// Mitsubishi GX Works2 project: finalfinal   PLC: FX3G

// global labels: Global1
VAR_GLOBAL
  workDayLight AT Y010 : BOOL;  (* Y010 is the work day light- lighting while the day running *)
  emergencyButton AT X007 : BOOL;  (* emergency button when click on the day stop *)
  startBlink AT M0 : BOOL;  (* when click on X007 -emergency button- the blinking function starts *)
  monitoringLighter AT M1 : BOOL;  (* monitoring light of the blinking *)
  timerBlink1 AT TC1 : BOOL;  (* timer for blink every 1 sec *)
  endTimerBlink1 AT TS1 : BOOL;  (* get value of 1 when TC1 is ending *)
END_VAR
VAR_GLOBAL CONSTANT
  timeBlink1 : INT := 10;
END_VAR
VAR_GLOBAL
  blinkLight1 AT M2 : BOOL;  (* one of the two lights that blinking in the blinking function that light Y010 blinking *)
  timerBlink2 AT TC2 : BOOL;  (* timer for blink every 1 sec *)
END_VAR
VAR_GLOBAL CONSTANT
  timeBlink2 : INT := 10;
END_VAR
VAR_GLOBAL
  endTimerBlink2 AT TS2 : BOOL;  (* get value of 1 when TC2  is ending *)
  blinkLight2 AT M3 : BOOL;  (* one of the blinking bulbs *)
END_VAR
VAR_GLOBAL CONSTANT
  initializeOrange : REAL := 170;  (* orange input for orit *)
END_VAR
VAR_GLOBAL
  startDayFictiveLight AT M4 : BOOL;  (* one condition of start the day- click on X010 start it *)
  stopAfter3Sec AT M5 : BOOL;  (* the light represent the end of 3 sec counting *)
END_VAR
VAR_GLOBAL CONSTANT
  count3Sec : INT := 600;
END_VAR
VAR_GLOBAL
  count3Sec2 AT TS3 : BOOL;  (* get 1 when TC3 ends after 3 sec *)
END_VAR
VAR_GLOBAL CONSTANT
  timer3Sec : INT := 30;
END_VAR
VAR_GLOBAL
  counter3Sec AT TC3 : BOOL;  (* 3 sec count for 2 bulbs blink 3 sec only and then stop *)
  orangeInput AT D1119 : REAL;  (* the amount of oranges we get for input *)
  OrangeQuantity AT D1121 : REAL;  (* moving orange input to our orange stack *)
  clementineInput AT D1123 : REAL;  (* the amount of clementine we get for input *)
  clementineQuantity AT D1125 : REAL;  (* moving clementine input to our clementine stack *)
  pomeloInput AT D1127 : REAL;  (* the amount of pomelo we get for input *)
  pomeloQuantity AT D1129 : REAL;  (* moving pomelo input to our pomelo stack *)
END_VAR
VAR_GLOBAL CONSTANT
  minOrange : REAL := 2.0;  (* check if we have at least 2 oranges unless the day cannot start *)
  minClementine : REAL := 1.0;  (* check if we have at least 1 clementine unless the day cannot start *)
  minPomelo : REAL := 1.0;  (* check if we have at least 1 pomelo unless the day cannot start *)
END_VAR
VAR_GLOBAL
  componentTesting AT M15 : BOOL;  (* if all the conditions are true the day can start *)
END_VAR
VAR_GLOBAL CONSTANT
  constantRatio : REAL := 2.0;  (* deviding or double orange in 2 *)
END_VAR
VAR_GLOBAL
  change AT D1133 : REAL;  (* the minimum of 0.5*orange, clementine, pomelo to use in the iteration *)
  changeOrange AT D1135 : REAL;  (* the real amount of orange we take to iteration *)
END_VAR
VAR_GLOBAL CONSTANT
  maxOrange : REAL := 50;  (* the max orange in iteration can be 100. so, if 0.5*orange is greater then 50 we take 50 *)
  value_1 : REAL := 1;
END_VAR
VAR_GLOBAL
  clemntineToUse AT D1137 : REAL;  (* move the chosen clementine value to use to the variable to use in the iteration *)
  pomeloToUse AT D1139 : REAL;  (* move the chosen pomelo value to use to the variable to use in the iteration *)
  orangeToUse AT D1141 : REAL;  (* move the chosen orange value to use to the variable to use in the iteration *)
  stratWashing AT X002 : BOOL;  (* start washing operation *)
  counter3secWash AT TC4 : BOOL;  (* count 3 sec of Y005 light in the wash operation *)
  washCounter3 AT TS4 : BOOL;  (* get 1 when TC4 3 sec ends *)
  stopLightWashing AT Y005 : BOOL;  (* washing light- light for 3 sec in the wash operation *)
  startWashing AT X002 : BOOL;  (* when part 1 is starting *)
  washingClemintine AT D1143 : REAL;  (* the clementine in the washing machine *)
  washingPomelo AT D1145 : REAL;  (* the pomelo in the washing machine *)
  washingOrange AT D1147 : REAL;  (* the orange in the washing machine *)
  squizeButton AT X001 : BOOL;  (* starts the squize operation *)
  squzeContainer AT D1149 : REAL;  (* all fruites dedicated to squize in the pre squize container *)
  finishWash AT M16 : BOOL;  (* represent the end of washing operation *)
  squizeLightStore AT Y001 : BOOL;  (* squize operation light- light until operation finish *)
  startSquize AT X011 : BOOL;  (* when push it twice the squize operatin starts *)
END_VAR
VAR_GLOBAL CONSTANT
  pushingCounter : INT := 2;
END_VAR
VAR_GLOBAL
  pushingCounterDevice AT CC0 : BOOL;  (* how much times we need to push to start squize *)
  doneCounter AT CS0 : BOOL;  (* when counter done finish squize *)
  squizeLight1 AT Y002 : BOOL;  (* blinking while squizing *)
  squizeLight2 AT Y003 : BOOL;  (* blinking while squizing *)
  emergencyButtonLight AT M8 : BOOL;  (* fictive light for emergency *)
  juiceContainer AT D1151 : REAL;  (* the juice container *)
  finishColectFruits AT M17 : BOOL;  (* when the colect ftuits is done the fictive lamp will light *)
  donesquizeLight AT M19 : BOOL;  (* squize ended *)
  startqualityCheck AT X003 : BOOL;  (* starts quality check operation *)
  startingQAcheckLight AT M20 : BOOL;  (* starting QA check Light *)
END_VAR
VAR_GLOBAL CONSTANT
  lowerBound : REAL := 1.0;  (* lower Bound *)
  upperBound : REAL := 5.0;  (* upper bound *)
END_VAR
VAR_GLOBAL
  timerOfQA AT TC6 : BOOL;  (* timer 5 sec of QA check *)
END_VAR
VAR_GLOBAL CONSTANT
  valueTimerQA : INT := 50;  (* valueTimerQA 5 SEC *)
END_VAR
VAR_GLOBAL
  doneTimerQA AT TS6 : BOOL;  (* when QA GOOD 5 sec light *)
  QAgoodLight AT Y004 : BOOL;  (* when QA GOOD 5 sec light Y005 *)
  stackcontainer AT D1155 : REAL;  (* stack Container *)
  analog_input_2 AT D8281 : INT;
  qualityChecking AT D1163 : REAL;  (* the quality check *)
  ifQAGood AT M22 : BOOL;  (* if QA good *)
  finishedQACheckLight AT M24 : BOOL;  (* when the good juice moved to stack the lamp will light *)
  juiceIsRotenLight AT M23 : BOOL;  (* when the qa check isnt good in the second time the juise is thrown out *)
  finishThrowJuiceLight AT M25 : BOOL;  (* when the roten juice is thrown out the lamp will light *)
  count2switchs AT CC1 : BOOL;  (* get 1 when X3 is up twice *)
END_VAR
VAR_GLOBAL CONSTANT
  twoSwitches : INT := 2;  (* 1 when there are 2 switch ups *)
END_VAR
VAR_GLOBAL
  counter2switches AT CS1 : BOOL;  (* 1 when 2 swiches happened *)
  startBottlingPart AT X005 : BOOL;  (* starts bottling part *)
  bottlingInProcessLight AT Y011 : BOOL;  (* the lamp will light till the bottling is in process *)
END_VAR
VAR_GLOBAL CONSTANT
  minNumOfLiters : REAL := 2.0;  (* check if we have at least 2 liter *)
  twoLittersInBottle : REAL := 2.0;  (* our buttles contains two litters *)
  maxBottles : REAL := 100.0;  (* the maximu bottles we can transfer *)
END_VAR
VAR_GLOBAL
  analog_output AT D8282 : INT;  (* analog value *)
END_VAR
VAR_GLOBAL CONSTANT
  normalizetion : REAL := 408;  (* analog value normalizetion *)
  normalizetion2 : REAL := 408;  (* analog value normalizetion *)
END_VAR
VAR_GLOBAL
  finishFirstBottling AT M6 : BOOL;  (* when the first bottling is done *)
  finishIteration AT Y006 : BOOL;  (* when the iteration is done *)
  timeBeforeSeceondTrack AT TC8 : BOOL;  (* stand still time before track num.2 *)
END_VAR
VAR_GLOBAL CONSTANT
  timeHold : INT := 20;
END_VAR
VAR_GLOBAL
  waitingSwitch AT TS8 : BOOL;  (* waiting for time to end to out track number 2 *)
  newStackContainer AT D1167 : REAL;
  updateInput AT M7 : BOOL;  (* update the input after every iteration *)
  endDay AT M9 : BOOL;  (* emergency button dtart the end day process *)
END_VAR
VAR_GLOBAL CONSTANT
  fourSecHolding : INT := 60;
END_VAR
VAR_GLOBAL
  trackDrivingFor4Sec2 AT TC10 : BOOL;  (* track light working for 4 sec *)
  trackDrivingTimer AT TS10 : BOOL;  (* track light working for 4 sec *)
  squizeStageLight AT X001 : BOOL;  (* squize operation light *)
  squizeStageLight2 AT M10 : BOOL;  (* squize operation light *)
  end5Stage AT M18 : BOOL;  (* indicte that the bottling process is done *)
  endOfBottlingPro AT M11 : BOOL;  (* indicte that the bottling process is done *)
END_VAR
VAR_GLOBAL CONSTANT
  minBottles : REAL := 1.0;  (* check if we have at least 1 clementine unless the day cannot start *)
  endOfBottle : REAL;  (* indicte that the bottling process is done *)
END_VAR
VAR_GLOBAL
  trackLight AT M12 : BOOL;  (* light of end track stage *)
  end5light AT M26 : BOOL;  (* indicte that the bottling process is done *)
  waitingBeforeExit AT TC9 : BOOL;  (* waiting for time to end to out track number 2 *)
  isWaitingOver AT TS9 : BOOL;  (* waiting for time to end to out track number 2 *)
  startSecondtrack AT X011 : BOOL;  (* when push it twice the squize operatin starts *)
  track2Timer AT TC10 : BOOL;  (* track light working for 4 sec *)
  track2Bool AT TS10 : BOOL;  (* track light working for 4 sec *)
  factiveBottlingLight AT M13 : BOOL;  (* gets 1 when bottling proccess start *)
  factiveQALight AT M21 : BOOL;  (* gets 1 when QA ends *)
END_VAR
VAR_GLOBAL CONSTANT
  zero : REAL;  (* zero value *)
END_VAR
VAR_GLOBAL
  factiveY5 AT M30 : BOOL;  (* when Y5 turn on *)
  factiveY1 AT M31 : BOOL;  (* when Y1 turn on *)
  tracl2bool AT TS10 : BOOL;  (* track light working for 4 sec *)
  stackcontainer2 AT D1165 : REAL;  (* stack Container *)
  moveToStackCon AT M27 : BOOL;  (* move stock to new container *)
  endDayZero AT M28 : BOOL;  (* if one of quantities is 0 the day over *)
  endDayZeroHold AT M29 : BOOL;  (* end Day Zero Hold STAY *)
  startDay AT X010 : BOOL;  (* the button for starting a work day *)
  numofBottles AT D1180 : REAL;  (* the new num of the bottles *)
  numofBottlesNew AT D1182 : REAL;  (* the new num of the bottles *)
  enoughFruit AT M37 : BOOL;  (* indicte that the GE function got 1 and there is enough fruits *)
  movingJuice AT M38 : BOOL;  (* end of moving juice into bottles *)
  analogOutput AT D1198 : REAL;  (* num of bottles for analog output *)
END_VAR

// task Task_01 (event TRUE, interval 0, priority 31): POU_01

PROGRAM POU_01
(* structured ladder/FBD written out as ST: instructions are called as NAME(EN, inputs, outputs); _pN, _eN, _tN stand for wires *)
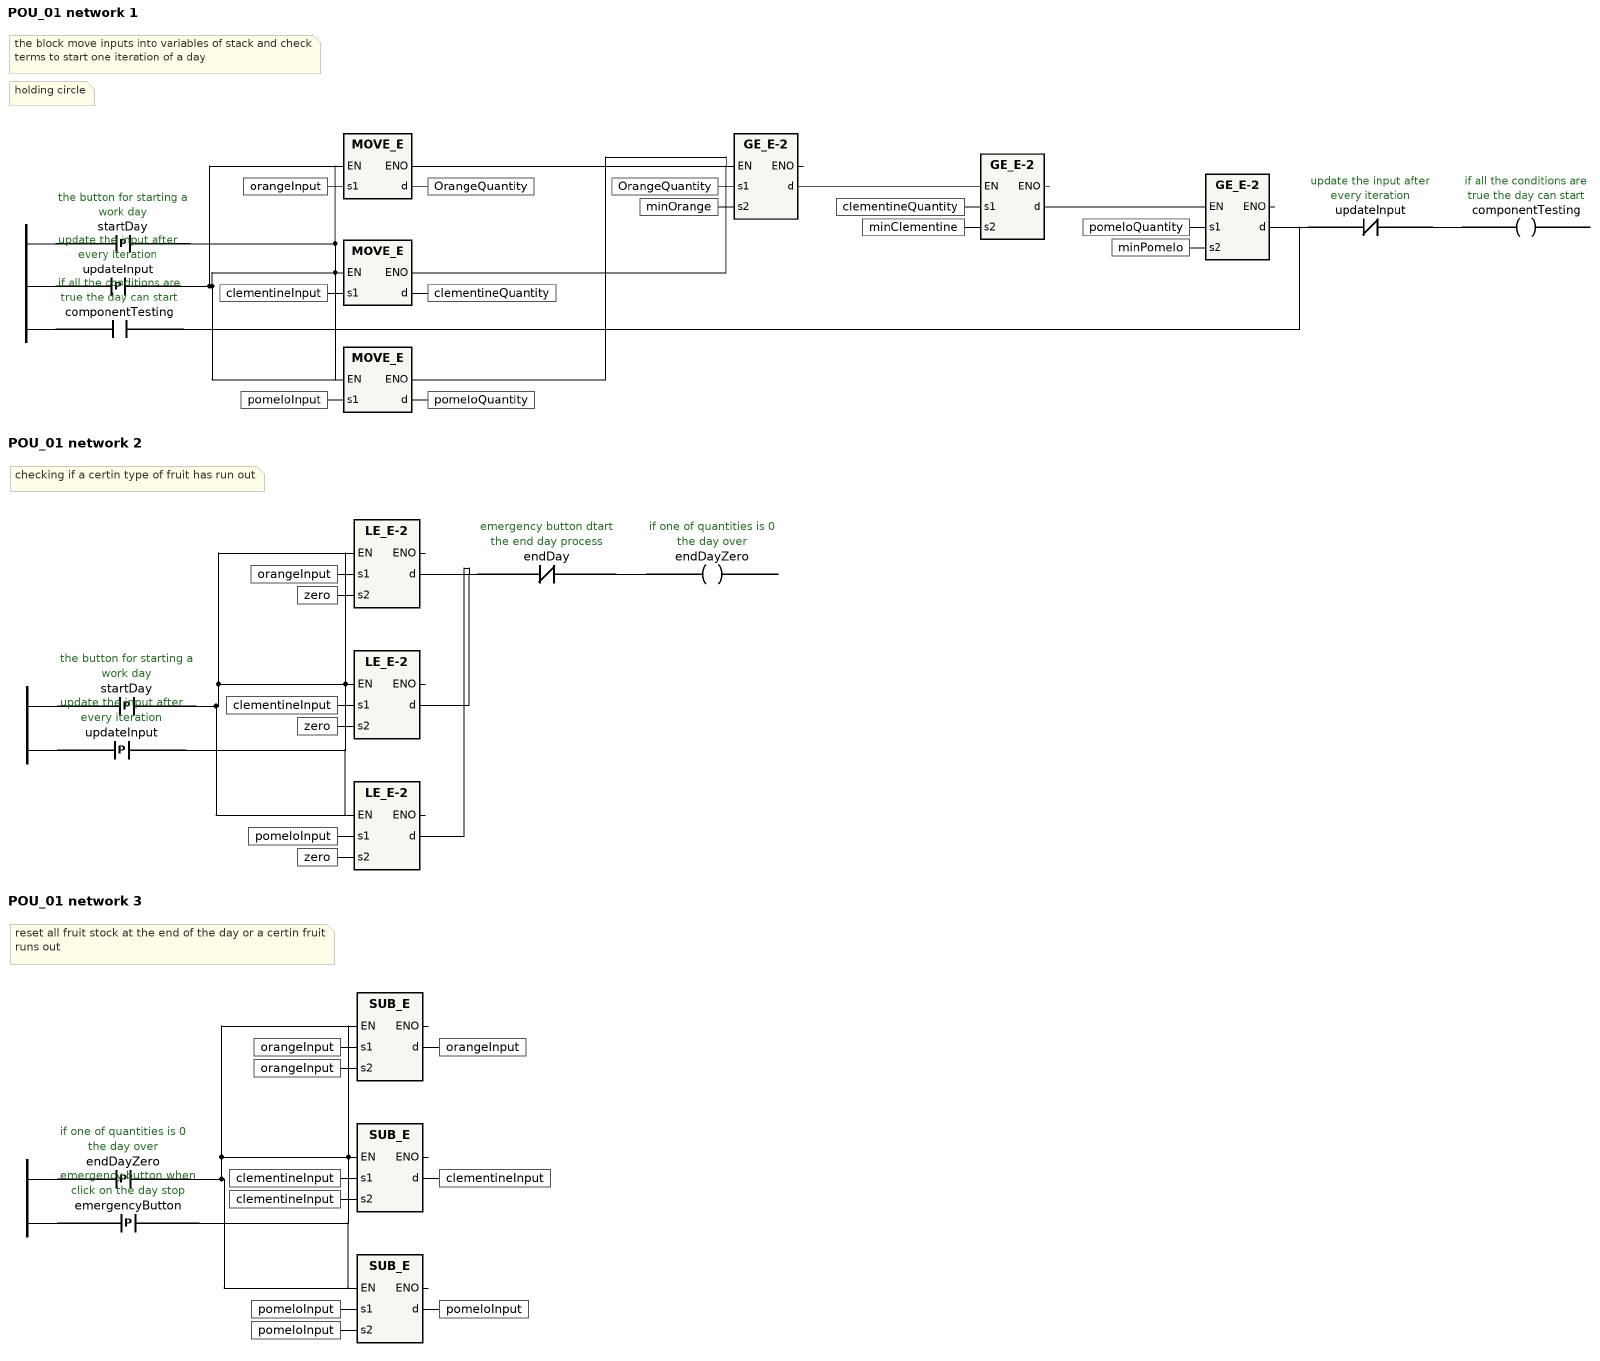
(* network 1 *)
(* the block move inputs into variables of stack and check terms to start one iteration of a day *)
(* holding circle *)
_p1 := LDP(TRUE, startDay) OR LDP(TRUE, updateInput);
_e2 := MOVE_E(_p1, orangeInput, OrangeQuantity);
_e3 := MOVE_E(_p1, clementineInput, clementineQuantity);
_e4 := MOVE_E(_p1, pomeloInput, pomeloQuantity);
GE_E(_e2 OR _e3 OR _e4, OrangeQuantity, minOrange, _t5);
GE_E(_t5, clementineQuantity, minClementine, _t6);
GE_E(_t6, pomeloQuantity, minPomelo, _t7);
componentTesting := (_t7 OR componentTesting) AND NOT updateInput;
(* network 2 *)
(* checking if a certin type of fruit has run out *)
_p1 := LDP(TRUE, startDay) OR LDP(TRUE, updateInput);
LE_E(_p1, orangeInput, zero, _t2);
LE_E(_p1, clementineInput, zero, _t3);
LE_E(_p1, pomeloInput, zero, _t4);
endDayZero := (_t2 OR _t3 OR _t4) AND NOT endDay;
(* network 3 *)
(* reset all fruit stock at the end of the day or a certin fruit runs out *)
_p1 := LDP(TRUE, endDayZero) OR LDP(TRUE, emergencyButton);
SUB_E(_p1, orangeInput, orangeInput, orangeInput);
SUB_E(_p1, clementineInput, clementineInput, clementineInput);
SUB_E(_p1, pomeloInput, pomeloInput, pomeloInput);
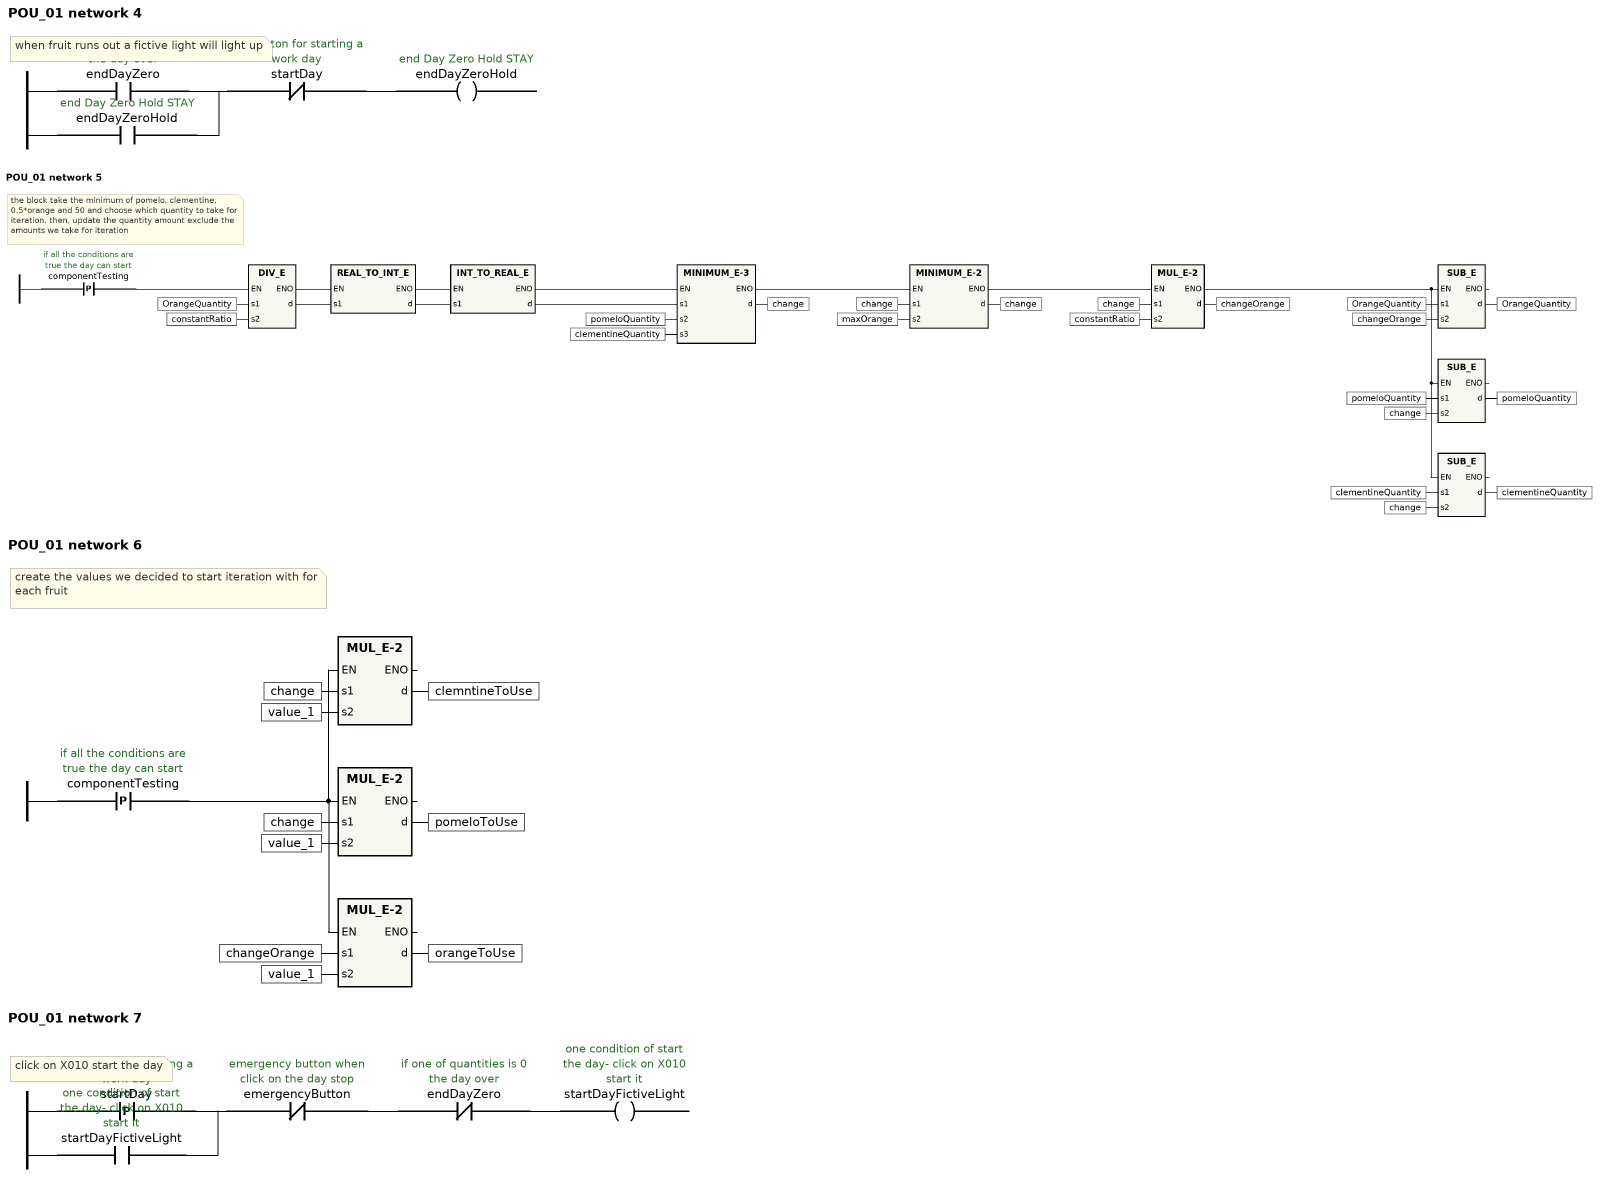
(* network 4 *)
(* when fruit runs out a fictive light will light up *)
endDayZeroHold := (endDayZero OR endDayZeroHold) AND NOT startDay;
(* network 5 *)
(* the block take the minimum of pomelo, clementine, 0.5*orange and 50 and choose which quantity to take for iteration. then, update the quantity amount exclude the amounts we take for iteration *)
_e2 := DIV_E(LDP(TRUE, componentTesting), OrangeQuantity, constantRatio, _t1);
_e4 := REAL_TO_INT_E(_e2, _t1, _t3);
_e6 := INT_TO_REAL_E(_e4, _t3, _t5);
_e7 := MINIMUM_E(_e6, _t5, pomeloQuantity, clementineQuantity, change);
_e8 := MINIMUM_E(_e7, change, maxOrange, change);
_e9 := MUL_E(_e8, change, constantRatio, changeOrange);
SUB_E(_e9, OrangeQuantity, changeOrange, OrangeQuantity);
SUB_E(_e9, pomeloQuantity, change, pomeloQuantity);
SUB_E(_e9, clementineQuantity, change, clementineQuantity);
(* network 6 *)
(* create the values we decided to start iteration with for each fruit *)
_p1 := LDP(TRUE, componentTesting);
MUL_E(_p1, change, value_1, clemntineToUse);
MUL_E(_p1, change, value_1, pomeloToUse);
MUL_E(_p1, changeOrange, value_1, orangeToUse);
(* network 7 *)
(* click on X010 start the day *)
startDayFictiveLight := ((LDP(TRUE, startDay) OR startDayFictiveLight) AND NOT emergencyButton) AND NOT endDayZero;
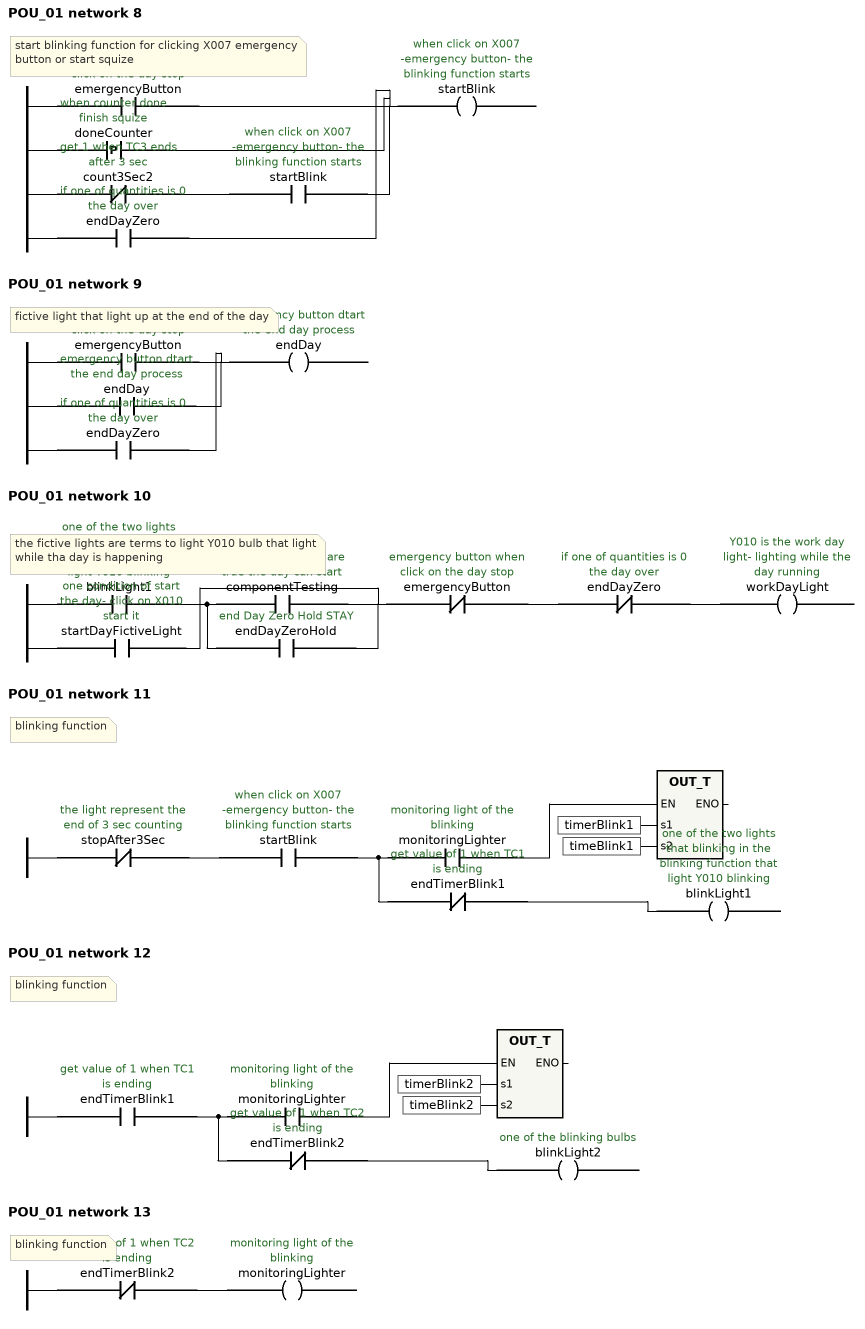
(* network 8 *)
(* start blinking function for clicking X007 emergency button or start squize *)
startBlink := emergencyButton OR LDP(TRUE, doneCounter) OR (NOT count3Sec2 AND startBlink) OR endDayZero;
(* network 9 *)
(* fictive light that light up at the end of the day *)
endDay := emergencyButton OR endDay OR endDayZero;
(* network 10 *)
(* the fictive lights are terms to light Y010 bulb that light while tha day is happening *)
workDayLight := (((blinkLight1 AND componentTesting) OR (blinkLight1 AND endDayZeroHold) OR startDayFictiveLight) AND NOT emergencyButton) AND NOT endDayZero;
(* network 11 *)
(* blinking function *)
_p1 := NOT stopAfter3Sec AND startBlink;
OUT_T(_p1 AND monitoringLighter, timerBlink1, timeBlink1);
blinkLight1 := _p1 AND NOT endTimerBlink1;
(* network 12 *)
(* blinking function *)
OUT_T(endTimerBlink1 AND monitoringLighter, timerBlink2, timeBlink2);
blinkLight2 := endTimerBlink1 AND NOT endTimerBlink2;
(* network 13 *)
(* blinking function *)
monitoringLighter := NOT endTimerBlink2;
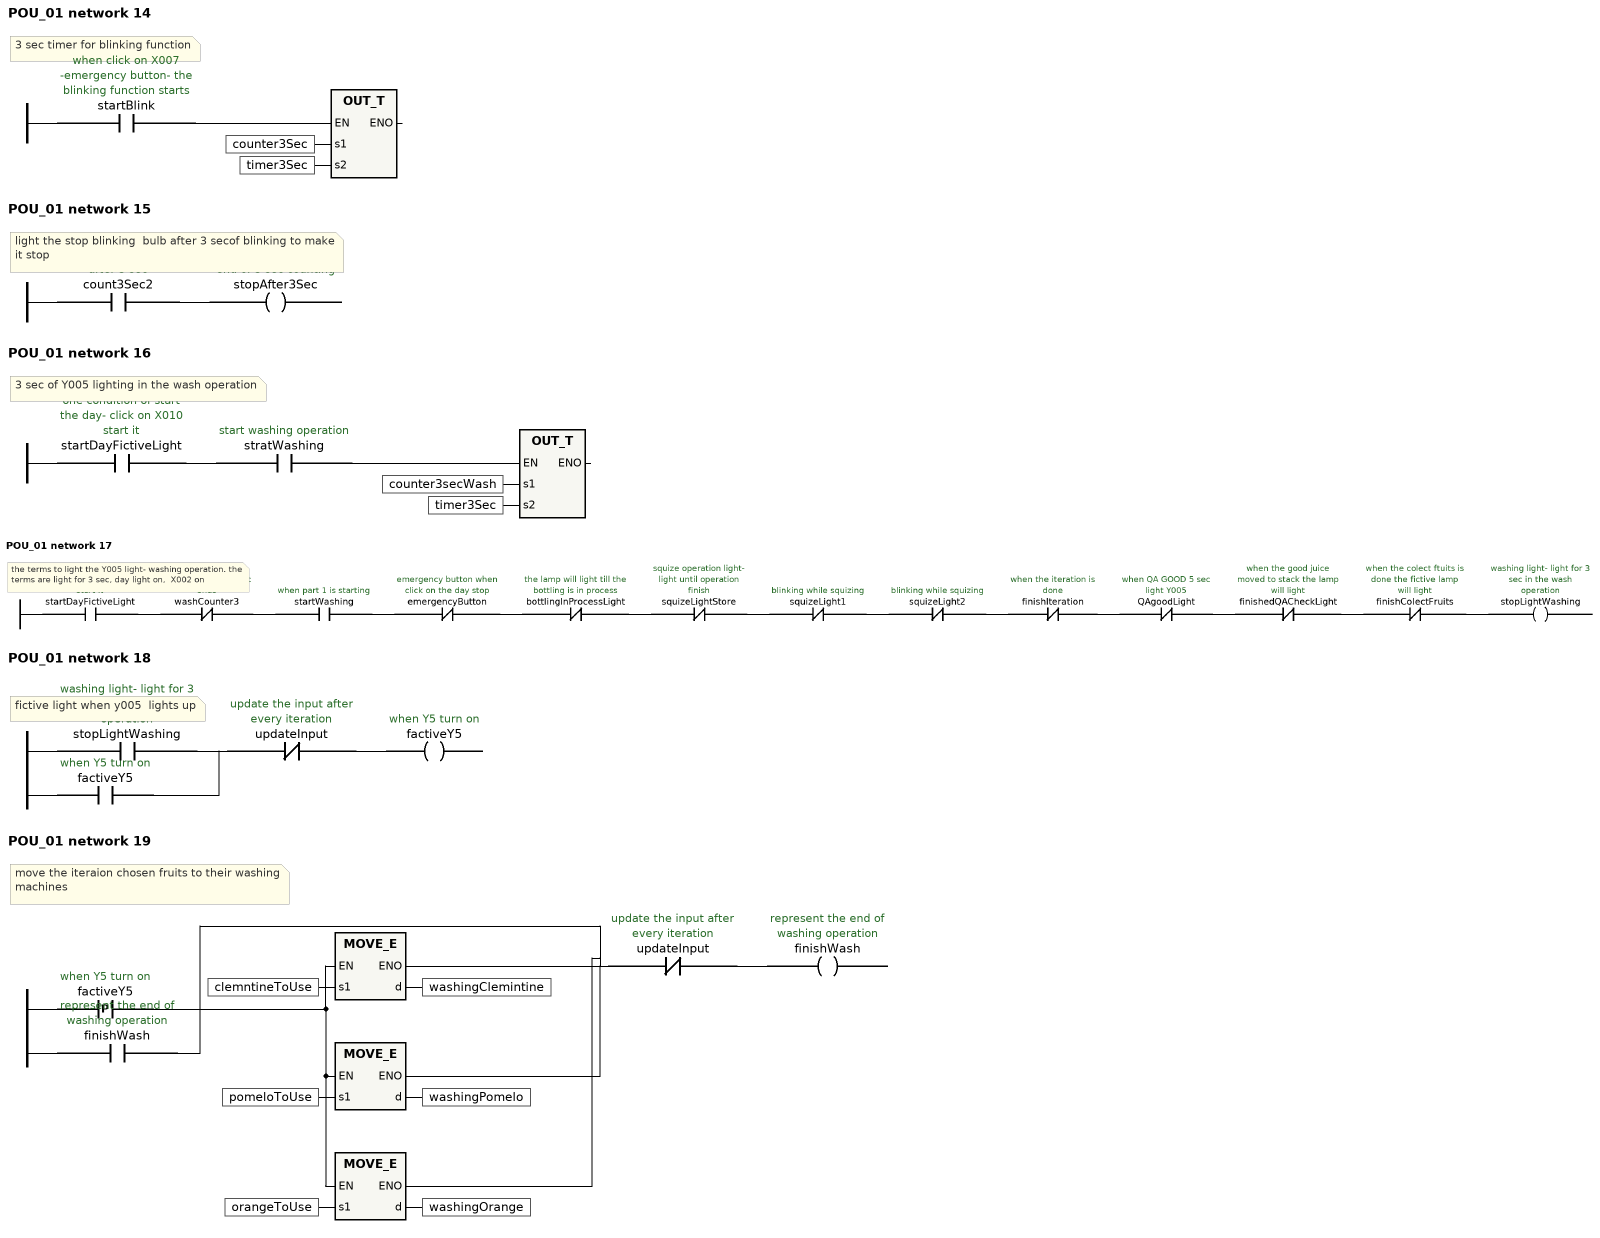
(* network 14 *)
(* 3 sec timer for blinking function *)
OUT_T(startBlink, counter3Sec, timer3Sec);
(* network 15 *)
(* light the stop blinking  bulb after 3 secof blinking to make it stop *)
stopAfter3Sec := count3Sec2;
(* network 16 *)
(* 3 sec of Y005 lighting in the wash operation *)
OUT_T(startDayFictiveLight AND stratWashing, counter3secWash, timer3Sec);
(* network 17 *)
(* the terms to light the Y005 light- washing operation. the terms are light for 3 sec, day light on,  X002 on *)
stopLightWashing := startDayFictiveLight AND NOT washCounter3 AND startWashing AND NOT emergencyButton AND NOT bottlingInProcessLight AND NOT squizeLightStore AND NOT squizeLight1 AND NOT squizeLight2 AND NOT finishIteration AND NOT QAgoodLight AND NOT finishedQACheckLight AND NOT finishColectFruits;
(* network 18 *)
(* fictive light when y005  lights up *)
factiveY5 := (stopLightWashing OR factiveY5) AND NOT updateInput;
(* network 19 *)
(* move the iteraion chosen fruits to their washing machines *)
_p1 := LDP(TRUE, factiveY5);
_e2 := MOVE_E(_p1, clemntineToUse, washingClemintine);
_e3 := MOVE_E(_p1, pomeloToUse, washingPomelo);
_e4 := MOVE_E(_p1, orangeToUse, washingOrange);
finishWash := (_e2 OR _e3 OR _e4 OR finishWash) AND NOT updateInput;
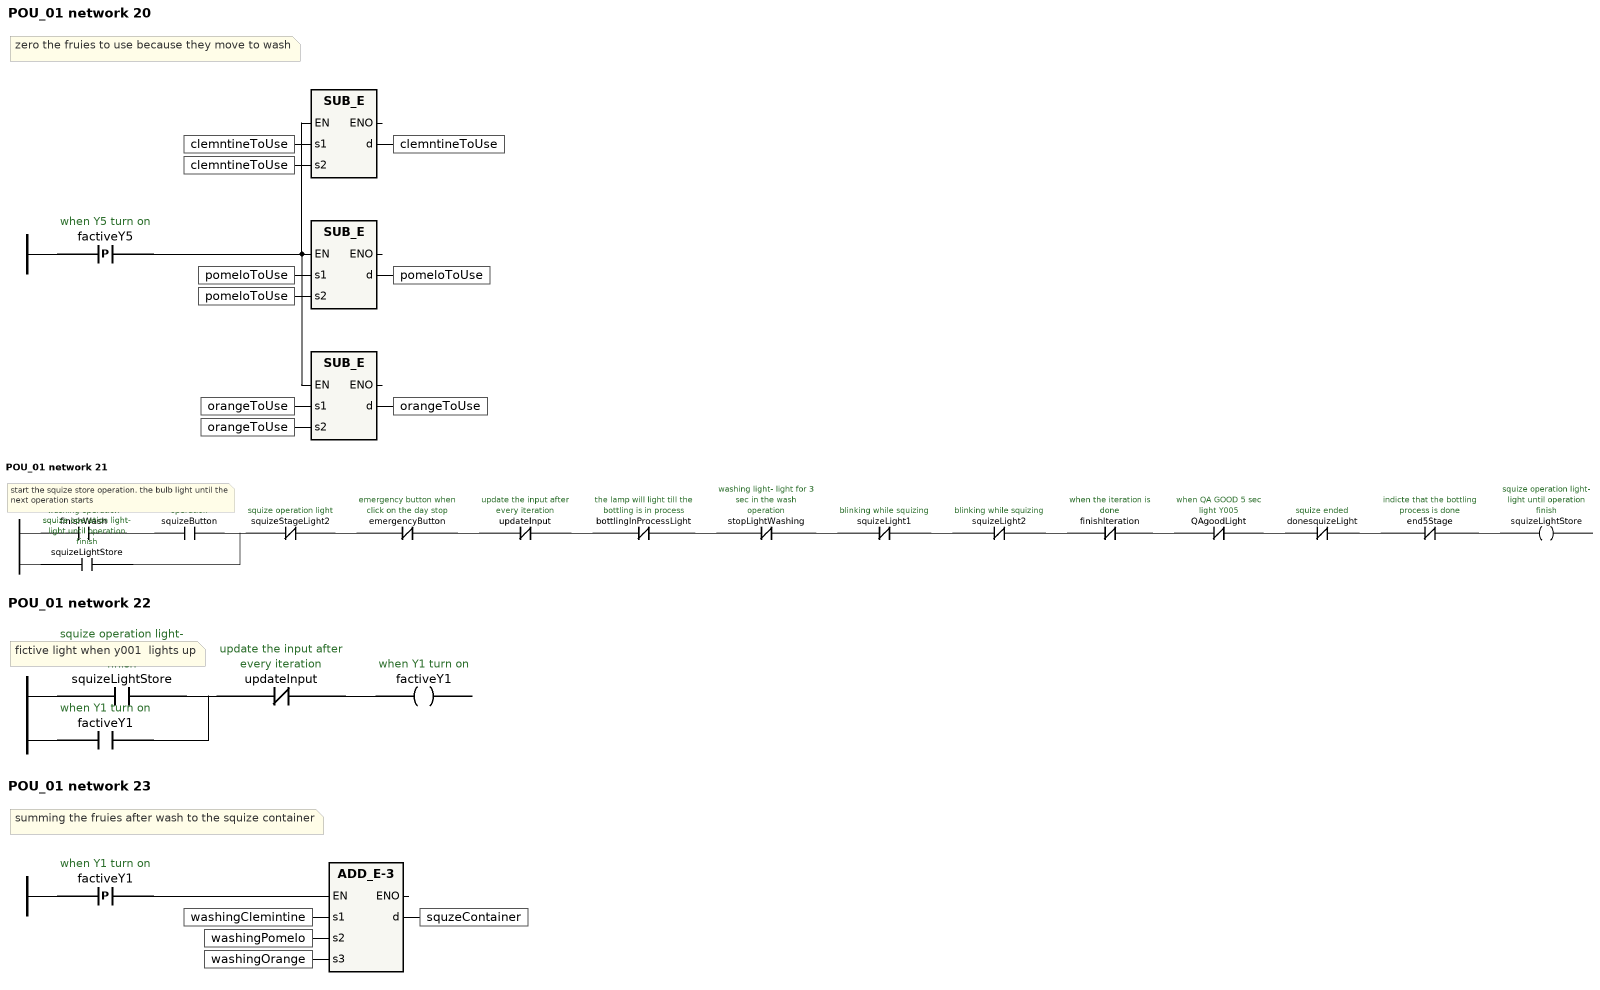
(* network 20 *)
(* zero the fruies to use because they move to wash *)
_p1 := LDP(TRUE, factiveY5);
SUB_E(_p1, clemntineToUse, clemntineToUse, clemntineToUse);
SUB_E(_p1, pomeloToUse, pomeloToUse, pomeloToUse);
SUB_E(_p1, orangeToUse, orangeToUse, orangeToUse);
(* network 21 *)
(* start the squize store operation. the bulb light until the next operation starts *)
squizeLightStore := ((((((((((((finishWash AND squizeButton) OR squizeLightStore) AND NOT squizeStageLight2) AND NOT emergencyButton) AND NOT updateInput) AND NOT bottlingInProcessLight) AND NOT stopLightWashing) AND NOT squizeLight1) AND NOT squizeLight2) AND NOT finishIteration) AND NOT QAgoodLight) AND NOT donesquizeLight) AND NOT end5Stage;
(* network 22 *)
(* fictive light when y001  lights up *)
factiveY1 := (squizeLightStore OR factiveY1) AND NOT updateInput;
(* network 23 *)
(* summing the fruies after wash to the squize container *)
ADD_E(LDP(TRUE, factiveY1), washingClemintine, washingPomelo, washingOrange, squzeContainer);
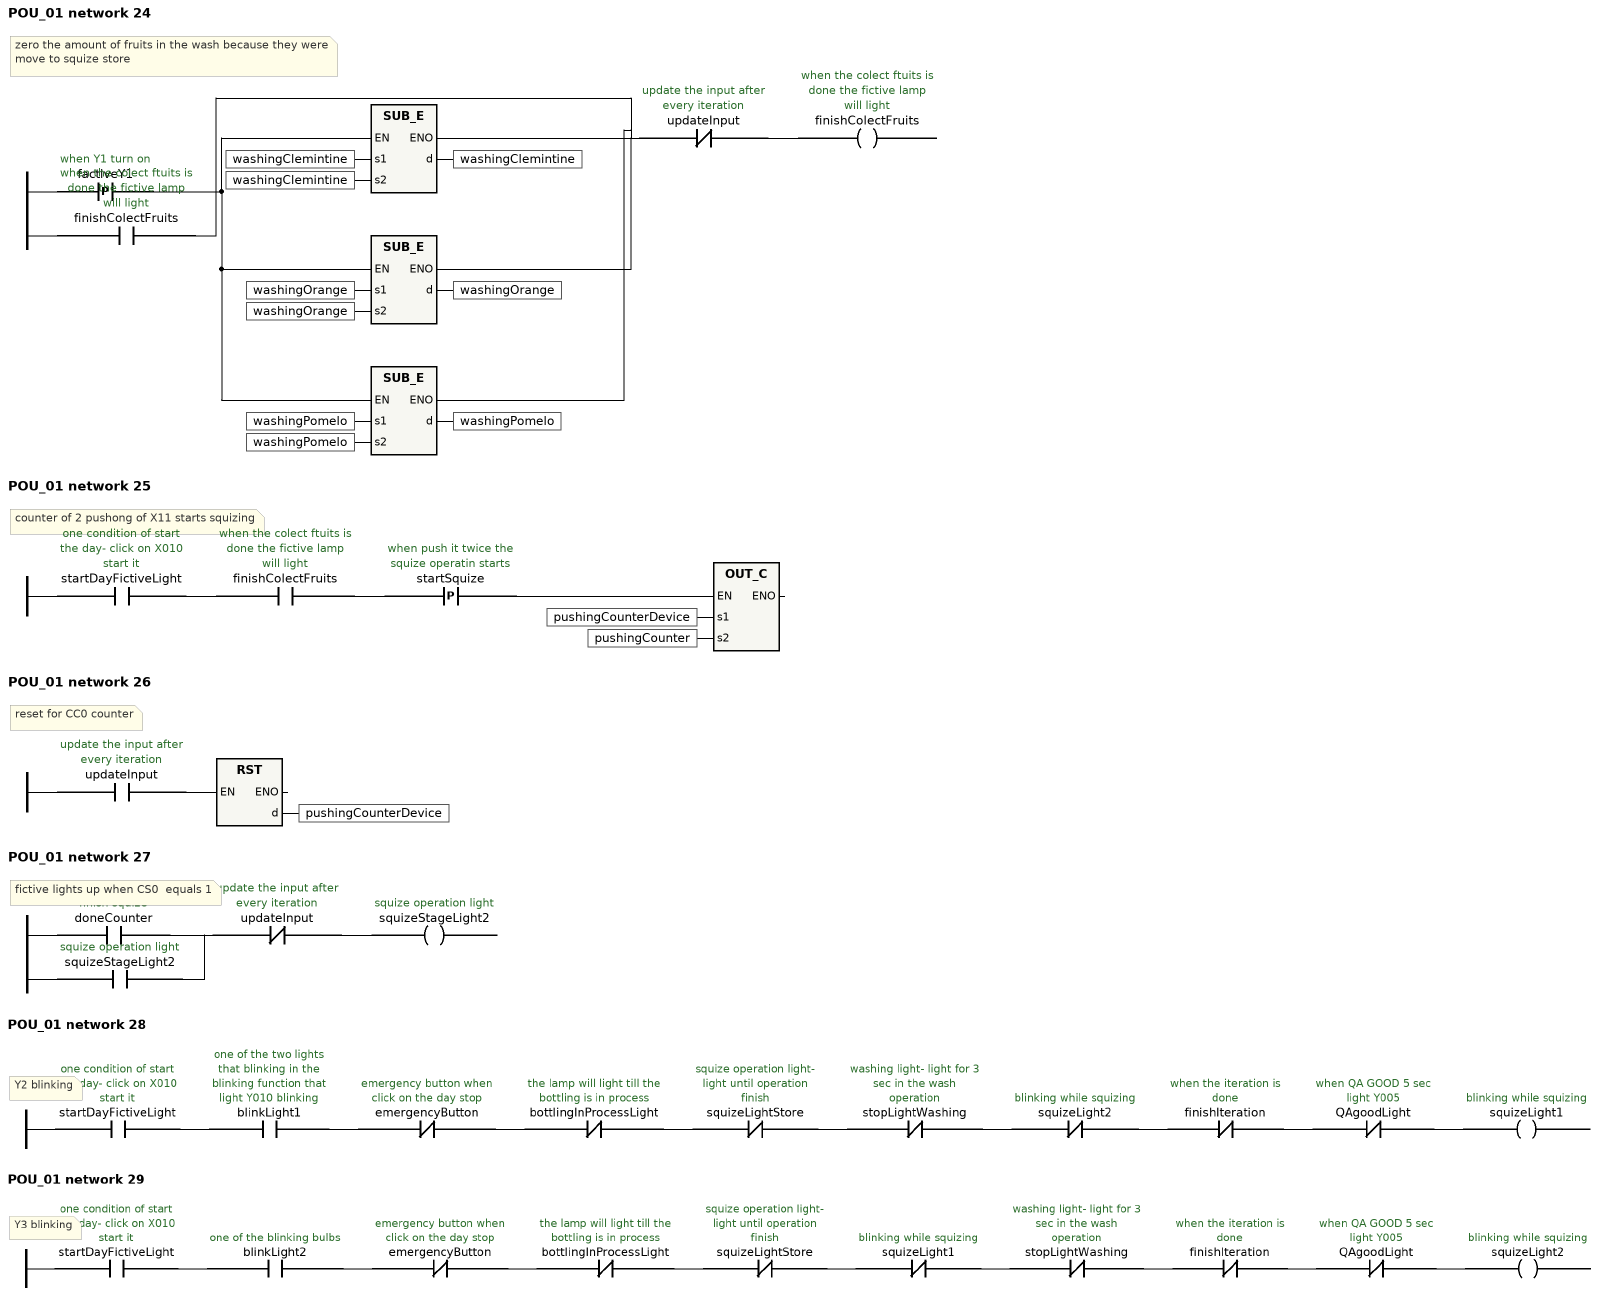
(* network 24 *)
(* zero the amount of fruits in the wash because they were move to squize store *)
_p1 := LDP(TRUE, factiveY1);
_e2 := SUB_E(_p1, washingClemintine, washingClemintine, washingClemintine);
_e3 := SUB_E(_p1, washingOrange, washingOrange, washingOrange);
_e4 := SUB_E(_p1, washingPomelo, washingPomelo, washingPomelo);
finishColectFruits := (_e2 OR _e3 OR _e4 OR finishColectFruits) AND NOT updateInput;
(* network 25 *)
(* counter of 2 pushong of X11 starts squizing *)
OUT_C(startDayFictiveLight AND finishColectFruits AND LDP(TRUE, startSquize), pushingCounterDevice, pushingCounter);
(* network 26 *)
(* reset for CC0 counter *)
RST(updateInput, pushingCounterDevice);
(* network 27 *)
(* fictive lights up when CS0  equals 1 *)
squizeStageLight2 := (doneCounter OR squizeStageLight2) AND NOT updateInput;
(* network 28 *)
(* Y2 blinking *)
squizeLight1 := startDayFictiveLight AND blinkLight1 AND NOT emergencyButton AND NOT bottlingInProcessLight AND NOT squizeLightStore AND NOT stopLightWashing AND NOT squizeLight2 AND NOT finishIteration AND NOT QAgoodLight;
(* network 29 *)
(* Y3 blinking *)
squizeLight2 := startDayFictiveLight AND blinkLight2 AND NOT emergencyButton AND NOT bottlingInProcessLight AND NOT squizeLightStore AND NOT squizeLight1 AND NOT stopLightWashing AND NOT finishIteration AND NOT QAgoodLight;
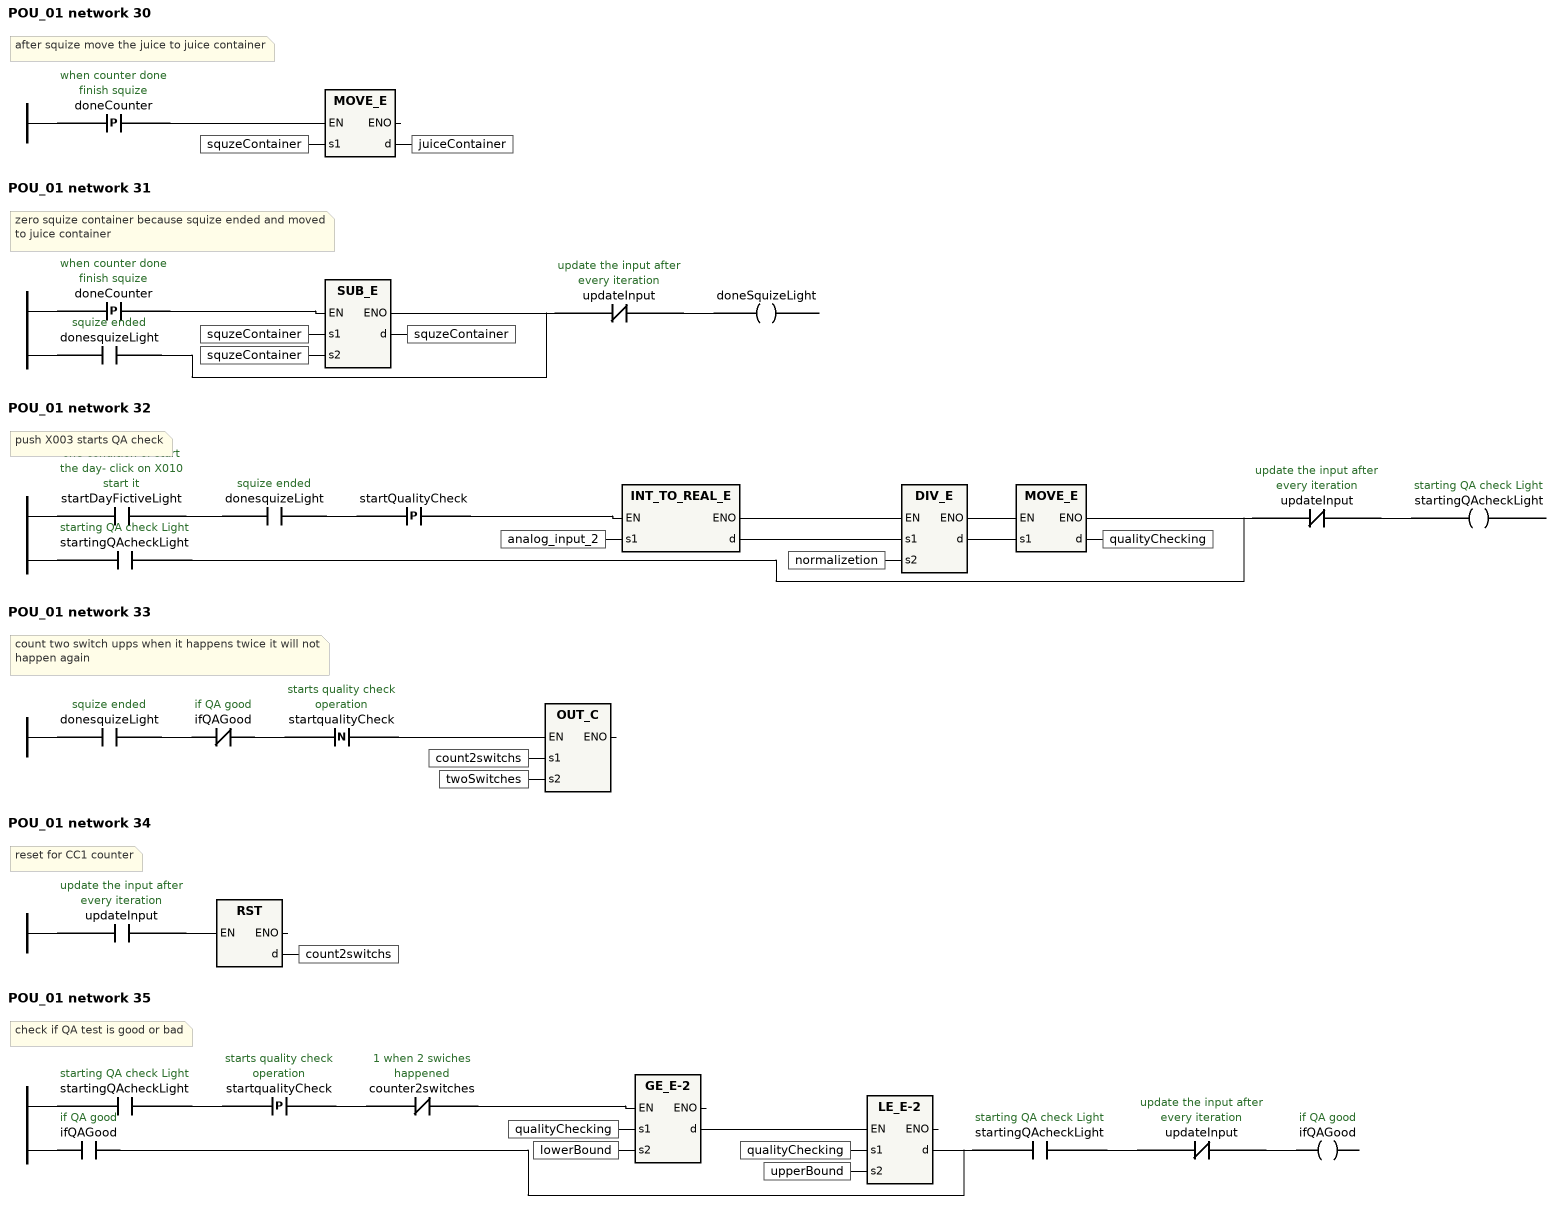
(* network 30 *)
(* after squize move the juice to juice container *)
MOVE_E(LDP(TRUE, doneCounter), squzeContainer, juiceContainer);
(* network 31 *)
(* zero squize container because squize ended and moved to juice container *)
_e1 := SUB_E(LDP(TRUE, doneCounter), squzeContainer, squzeContainer, squzeContainer);
doneSquizeLight := (_e1 OR donesquizeLight) AND NOT updateInput;
(* network 32 *)
(* push X003 starts QA check *)
_e2 := INT_TO_REAL_E(startDayFictiveLight AND donesquizeLight AND LDP(TRUE, startQualityCheck), analog_input_2, _t1);
_e4 := DIV_E(_e2, _t1, normalizetion, _t3);
_e5 := MOVE_E(_e4, _t3, qualityChecking);
startingQAcheckLight := (_e5 OR startingQAcheckLight) AND NOT updateInput;
(* network 33 *)
(* count two switch upps when it happens twice it will not happen again *)
OUT_C(donesquizeLight AND NOT ifQAGood AND LDF(TRUE, startqualityCheck), count2switchs, twoSwitches);
(* network 34 *)
(* reset for CC1 counter *)
RST(updateInput, count2switchs);
(* network 35 *)
(* check if QA test is good or bad *)
GE_E(startingQAcheckLight AND LDP(TRUE, startqualityCheck) AND NOT counter2switches, qualityChecking, lowerBound, _t1);
LE_E(_t1, qualityChecking, upperBound, _t2);
ifQAGood := ((_t2 OR ifQAGood) AND startingQAcheckLight) AND NOT updateInput;
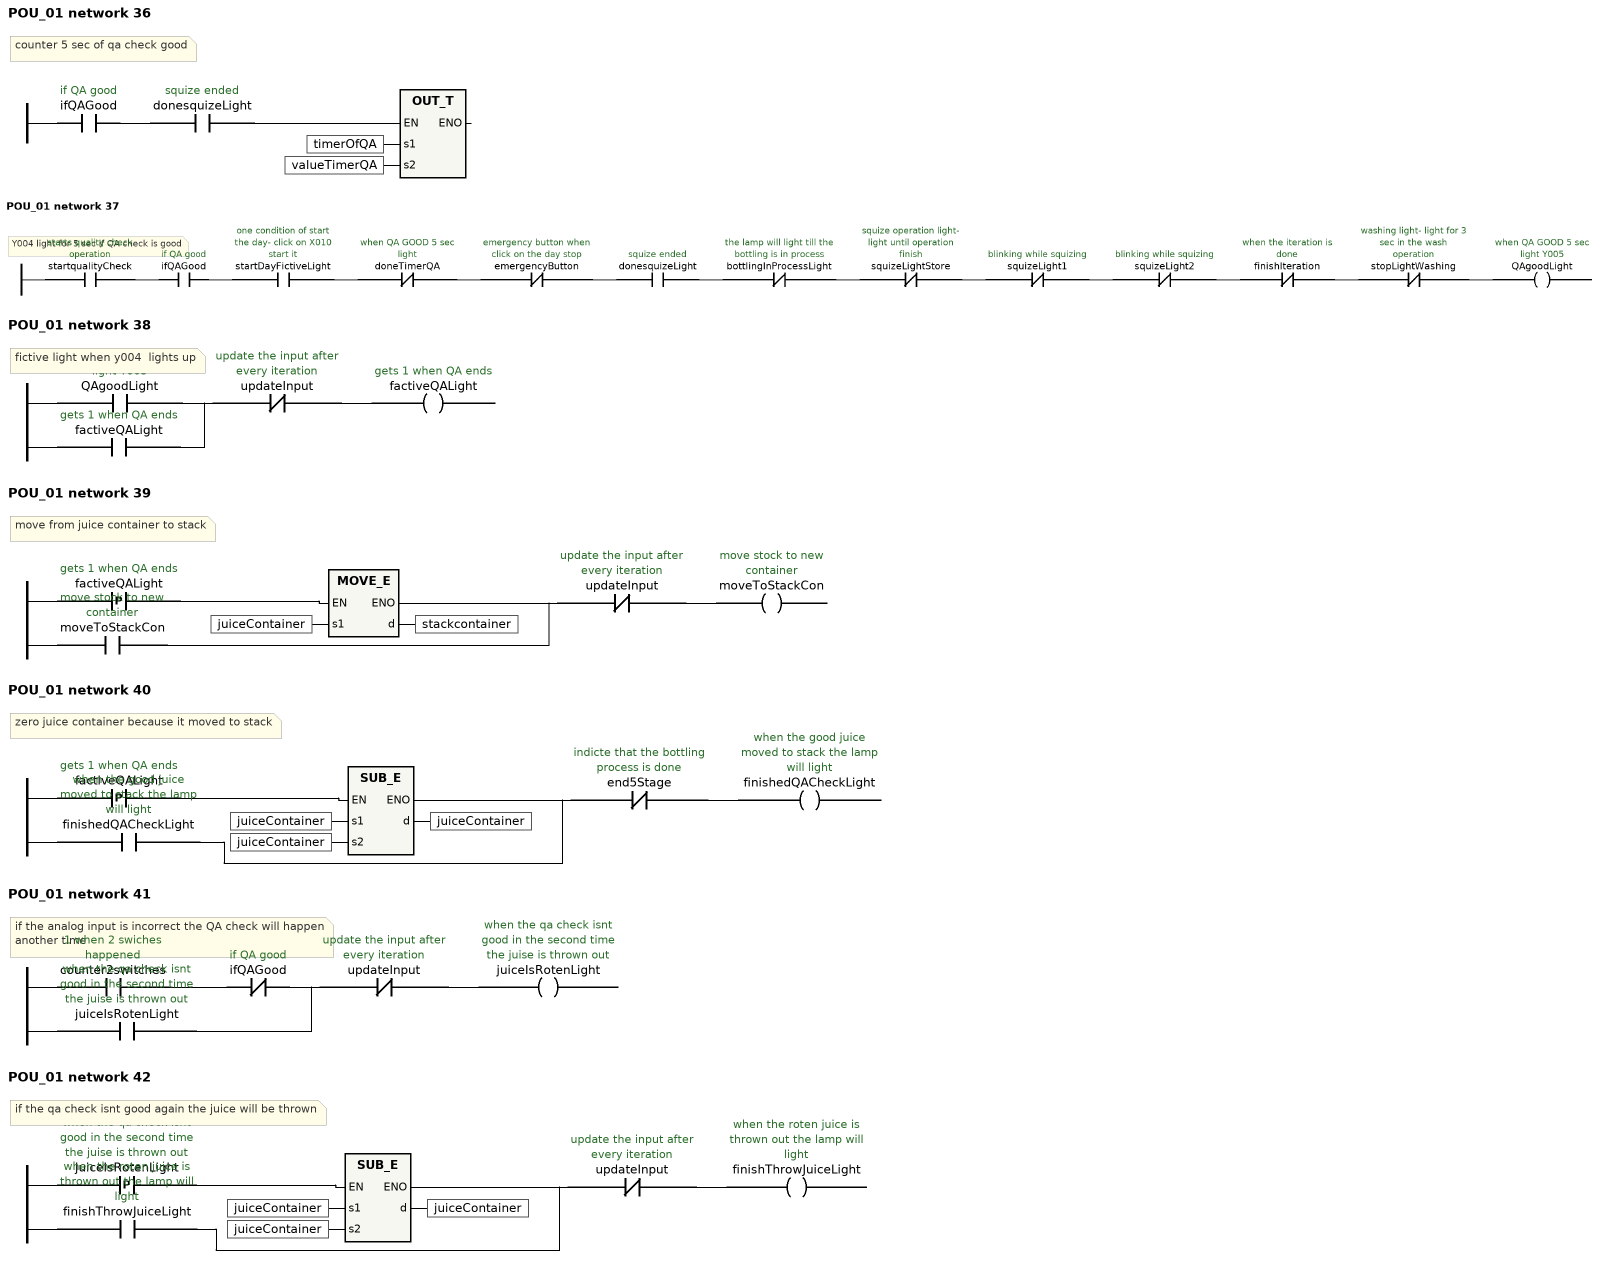
(* network 36 *)
(* counter 5 sec of qa check good *)
OUT_T(ifQAGood AND donesquizeLight, timerOfQA, valueTimerQA);
(* network 37 *)
(* Y004 light for 5 sec if QA check is good *)
QAgoodLight := startqualityCheck AND ifQAGood AND startDayFictiveLight AND NOT doneTimerQA AND NOT emergencyButton AND donesquizeLight AND NOT bottlingInProcessLight AND NOT squizeLightStore AND NOT squizeLight1 AND NOT squizeLight2 AND NOT finishIteration AND NOT stopLightWashing;
(* network 38 *)
(* fictive light when y004  lights up *)
factiveQALight := (QAgoodLight OR factiveQALight) AND NOT updateInput;
(* network 39 *)
(* move from juice container to stack *)
_e1 := MOVE_E(LDP(TRUE, factiveQALight), juiceContainer, stackcontainer);
moveToStackCon := (_e1 OR moveToStackCon) AND NOT updateInput;
(* network 40 *)
(* zero juice container because it moved to stack *)
_e1 := SUB_E(LDP(TRUE, factiveQALight), juiceContainer, juiceContainer, juiceContainer);
finishedQACheckLight := (_e1 OR finishedQACheckLight) AND NOT end5Stage;
(* network 41 *)
(* if the analog input is incorrect the QA check will happen another time *)
juiceIsRotenLight := ((counter2switches AND NOT ifQAGood) OR juiceIsRotenLight) AND NOT updateInput;
(* network 42 *)
(* if the qa check isnt good again the juice will be thrown *)
_e1 := SUB_E(LDP(TRUE, juiceIsRotenLight), juiceContainer, juiceContainer, juiceContainer);
finishThrowJuiceLight := (_e1 OR finishThrowJuiceLight) AND NOT updateInput;
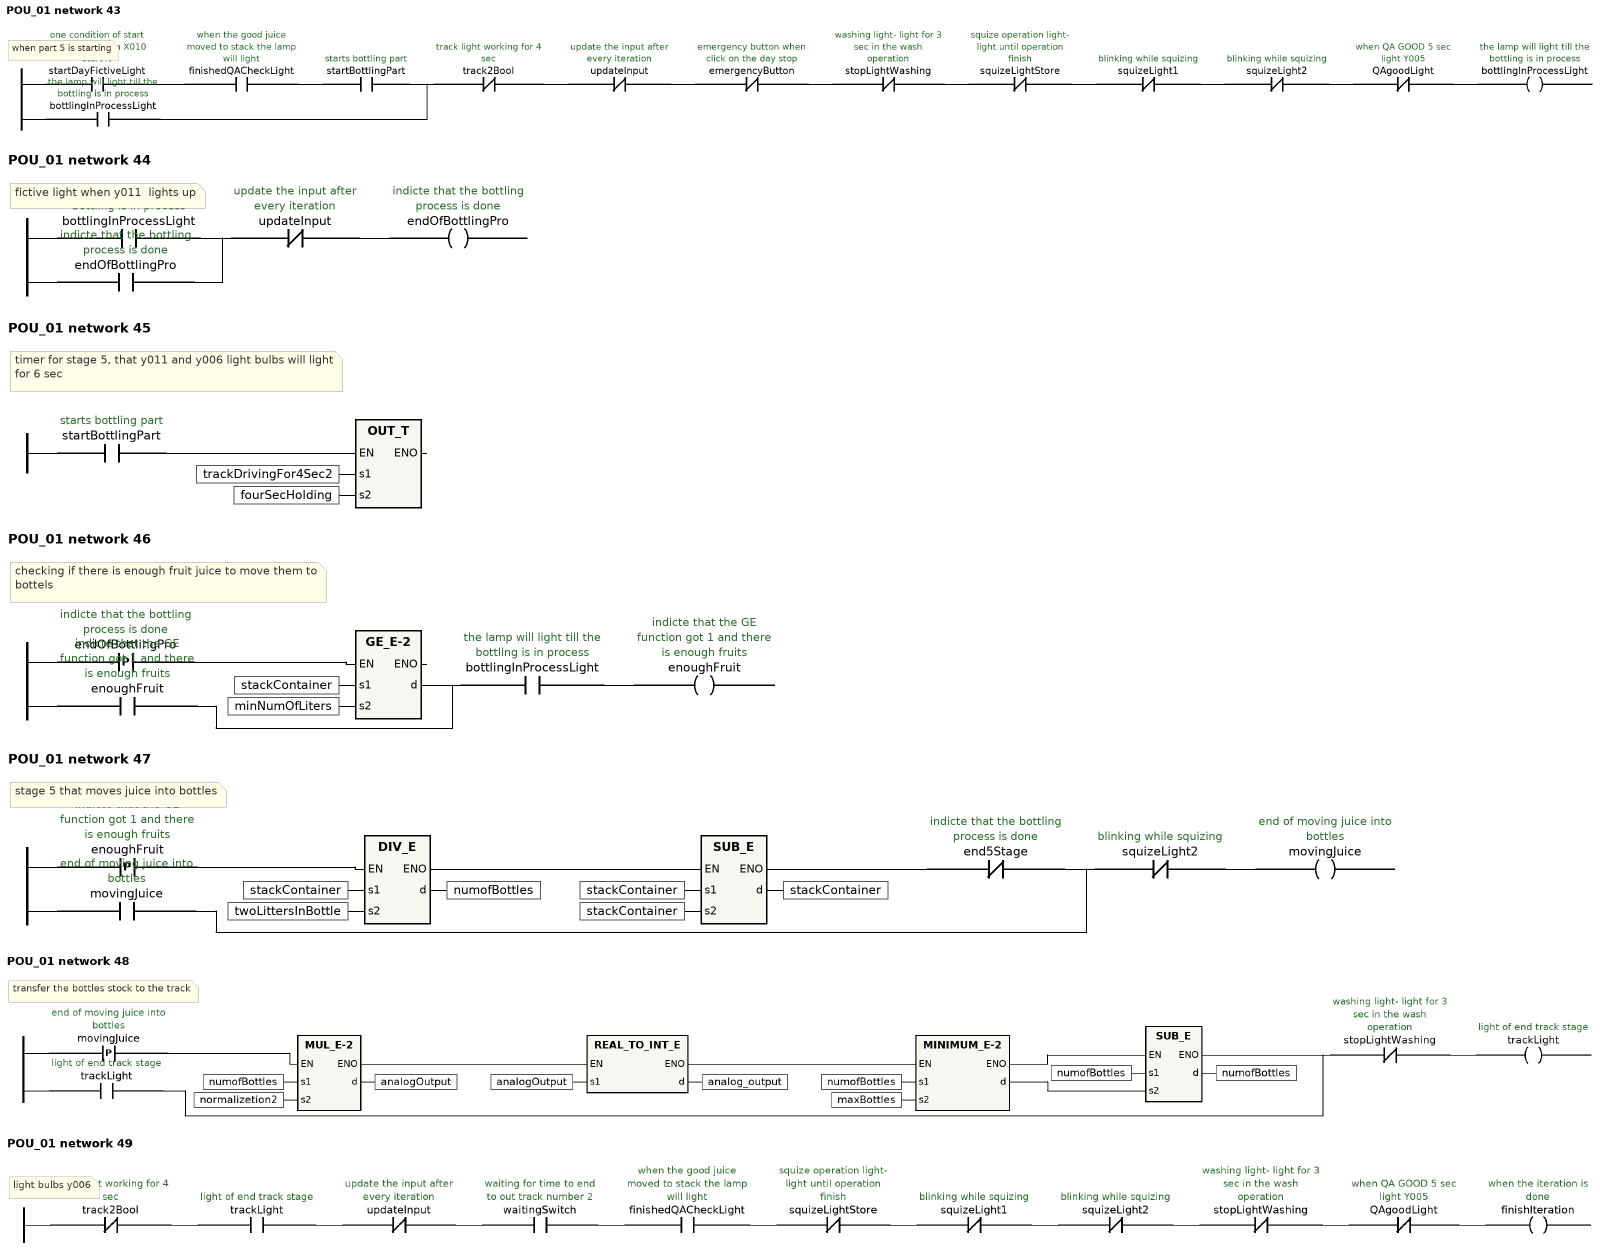
(* network 43 *)
(* when part 5 is starting *)
bottlingInProcessLight := (((((((((startDayFictiveLight AND finishedQACheckLight AND startBottlingPart) OR bottlingInProcessLight) AND NOT track2Bool) AND NOT updateInput) AND NOT emergencyButton) AND NOT stopLightWashing) AND NOT squizeLightStore) AND NOT squizeLight1) AND NOT squizeLight2) AND NOT QAgoodLight;
(* network 44 *)
(* fictive light when y011  lights up *)
endOfBottlingPro := (bottlingInProcessLight OR endOfBottlingPro) AND NOT updateInput;
(* network 45 *)
(* timer for stage 5, that y011 and y006 light bulbs will light for 6 sec *)
OUT_T(startBottlingPart, trackDrivingFor4Sec2, fourSecHolding);
(* network 46 *)
(* checking if there is enough fruit juice to move them to bottels *)
GE_E(LDP(TRUE, endOfBottlingPro), stackContainer, minNumOfLiters, _t1);
enoughFruit := (_t1 OR enoughFruit) AND bottlingInProcessLight;
(* network 47 *)
(* stage 5 that moves juice into bottles *)
_e1 := DIV_E(LDP(TRUE, enoughFruit), stackContainer, twoLittersInBottle, numofBottles);
_e2 := SUB_E(_e1, stackContainer, stackContainer, stackContainer);
movingJuice := ((_e2 AND NOT end5Stage) OR movingJuice) AND NOT squizeLight2;
(* network 48 *)
(* transfer the bottles stock to the track *)
_e1 := MUL_E(LDP(TRUE, movingJuice), numofBottles, normalizetion2, analogOutput);
_e2 := REAL_TO_INT_E(_e1, analogOutput, analog_output);
_e4 := MINIMUM_E(_e2, numofBottles, maxBottles, _t3);
_e5 := SUB_E(_e4, numofBottles, _t3, numofBottles);
trackLight := (_e5 OR trackLight) AND NOT stopLightWashing;
(* network 49 *)
(* light bulbs y006 *)
finishIteration := NOT track2Bool AND trackLight AND NOT updateInput AND waitingSwitch AND finishedQACheckLight AND NOT squizeLightStore AND NOT squizeLight1 AND NOT squizeLight2 AND NOT stopLightWashing AND NOT QAgoodLight;
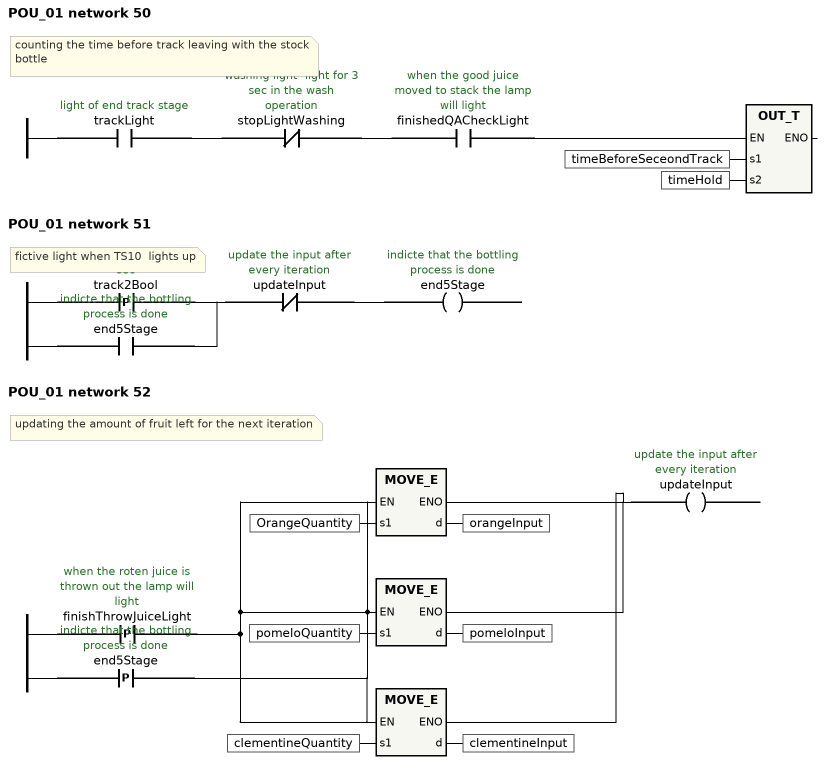
(* network 50 *)
(* counting the time before track leaving with the stock bottle *)
OUT_T(trackLight AND NOT stopLightWashing AND finishedQACheckLight, timeBeforeSeceondTrack, timeHold);
(* network 51 *)
(* fictive light when TS10  lights up *)
end5Stage := (LDP(TRUE, track2Bool) OR end5Stage) AND NOT updateInput;
(* network 52 *)
(* updating the amount of fruit left for the next iteration *)
_p1 := LDP(TRUE, finishThrowJuiceLight) OR LDP(TRUE, end5Stage);
_e2 := MOVE_E(_p1, OrangeQuantity, orangeInput);
_e3 := MOVE_E(_p1, pomeloQuantity, pomeloInput);
_e4 := MOVE_E(_p1, clementineQuantity, clementineInput);
updateInput := _e2 OR _e3 OR _e4;
END_PROGRAM
